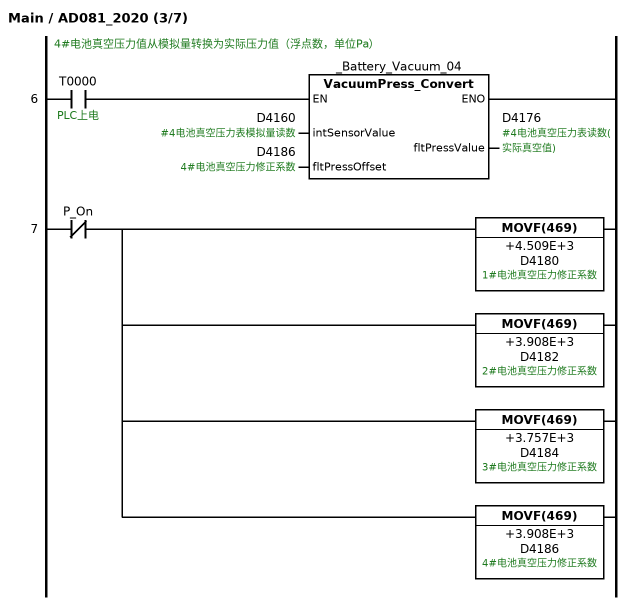
; [picture p24: Main / AD081_2020, rungs 6-7]
; rung 6: 4#电池真空压力值从模拟量转换为实际压力值（浮点数，单位Pa）
LD T0000  ; PLC上电
CALL _Battery_Vacuum_04 : VacuumPress_Convert (intSensorValue := D4160, fltPressOffset := D4186, fltPressValue => D4176)  ; #4电池真空压力表模拟量读数, 4#电池真空压力修正系数, #4电池真空压力表读数(实际真空值)
; rung 7
LDNOT P_On
MOVF(469) +4.509E+3 D4180  ; 1#电池真空压力修正系数
MOVF(469) +3.908E+3 D4182  ; 2#电池真空压力修正系数
MOVF(469) +3.757E+3 D4184  ; 3#电池真空压力修正系数
MOVF(469) +3.908E+3 D4186  ; 4#电池真空压力修正系数

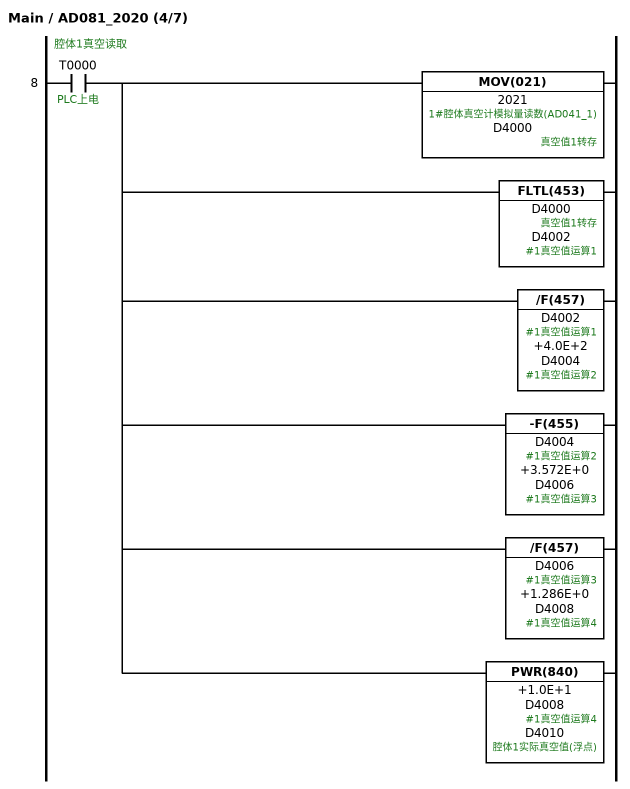
; rung 8: 腔体1真空读取
LD T0000  ; PLC上电
MOV(021) 2021 D4000  ; 1#腔体真空计模拟量读数(AD041_1), 真空值1转存
FLTL(453) D4000 D4002  ; 真空值1转存, #1真空值运算1
/F(457) D4002 +4.0E+2 D4004  ; #1真空值运算1, #1真空值运算2
-F(455) D4004 +3.572E+0 D4006  ; #1真空值运算2, #1真空值运算3
/F(457) D4006 +1.286E+0 D4008  ; #1真空值运算3, #1真空值运算4
PWR(840) +1.0E+1 D4008 D4010  ; #1真空值运算4, 腔体1实际真空值(浮点)

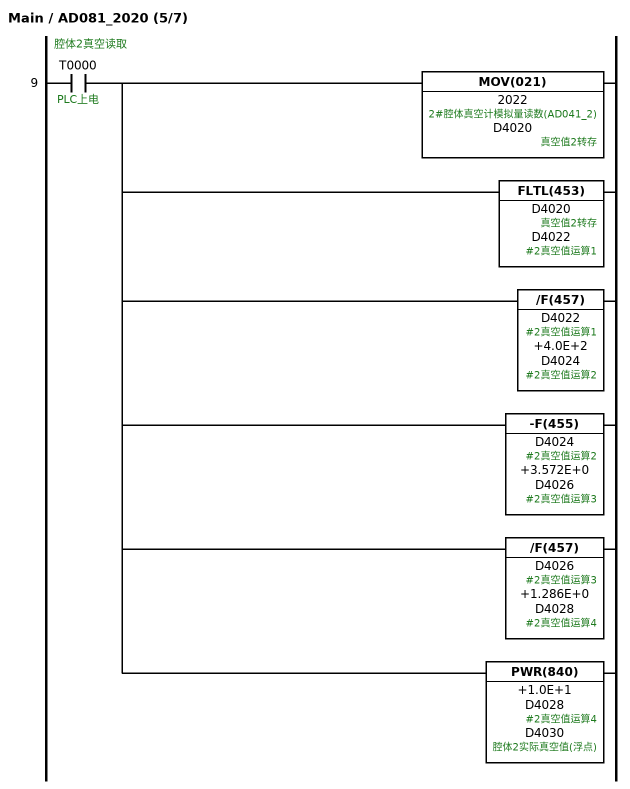
; rung 9: 腔体2真空读取
LD T0000  ; PLC上电
MOV(021) 2022 D4020  ; 2#腔体真空计模拟量读数(AD041_2), 真空值2转存
FLTL(453) D4020 D4022  ; 真空值2转存, #2真空值运算1
/F(457) D4022 +4.0E+2 D4024  ; #2真空值运算1, #2真空值运算2
-F(455) D4024 +3.572E+0 D4026  ; #2真空值运算2, #2真空值运算3
/F(457) D4026 +1.286E+0 D4028  ; #2真空值运算3, #2真空值运算4
PWR(840) +1.0E+1 D4028 D4030  ; #2真空值运算4, 腔体2实际真空值(浮点)

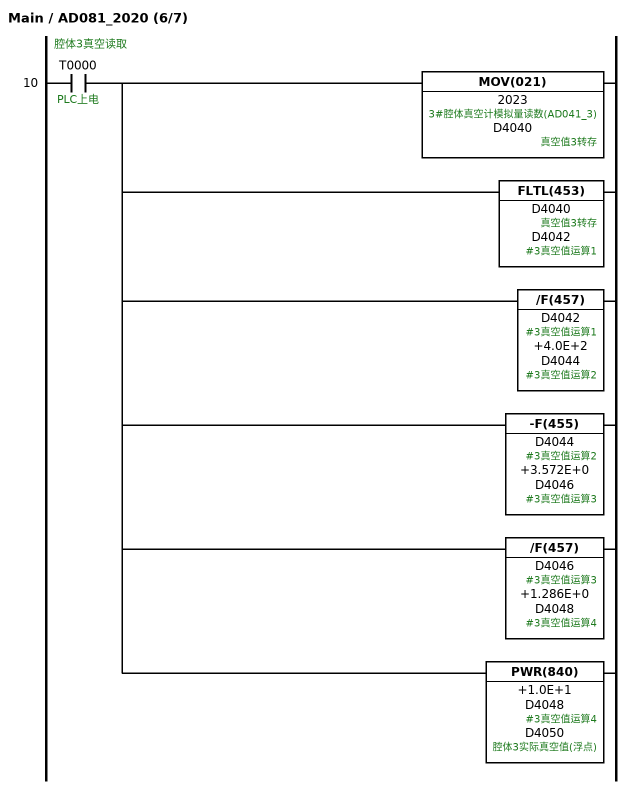
; rung 10: 腔体3真空读取
LD T0000  ; PLC上电
MOV(021) 2023 D4040  ; 3#腔体真空计模拟量读数(AD041_3), 真空值3转存
FLTL(453) D4040 D4042  ; 真空值3转存, #3真空值运算1
/F(457) D4042 +4.0E+2 D4044  ; #3真空值运算1, #3真空值运算2
-F(455) D4044 +3.572E+0 D4046  ; #3真空值运算2, #3真空值运算3
/F(457) D4046 +1.286E+0 D4048  ; #3真空值运算3, #3真空值运算4
PWR(840) +1.0E+1 D4048 D4050  ; #3真空值运算4, 腔体3实际真空值(浮点)

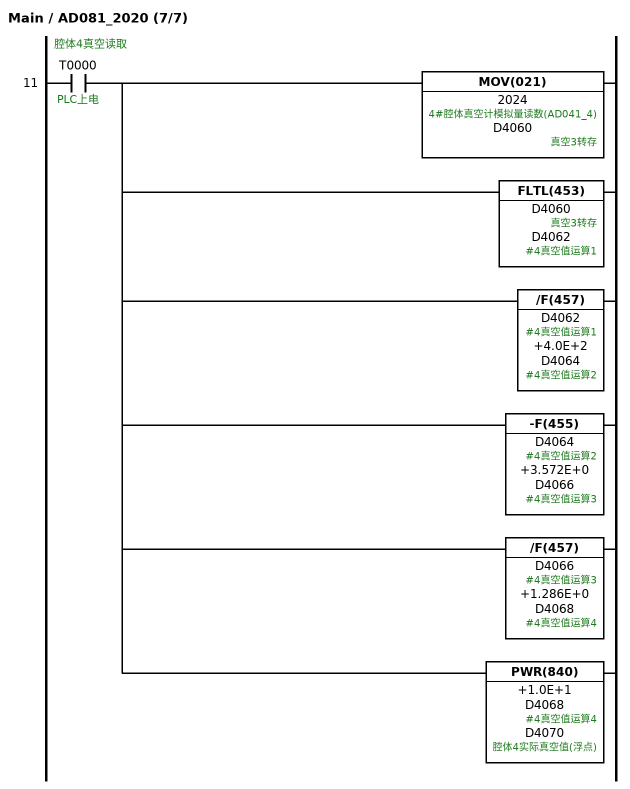
; rung 11: 腔体4真空读取
LD T0000  ; PLC上电
MOV(021) 2024 D4060  ; 4#腔体真空计模拟量读数(AD041_4), 真空3转存
FLTL(453) D4060 D4062  ; 真空3转存, #4真空值运算1
/F(457) D4062 +4.0E+2 D4064  ; #4真空值运算1, #4真空值运算2
-F(455) D4064 +3.572E+0 D4066  ; #4真空值运算2, #4真空值运算3
/F(457) D4066 +1.286E+0 D4068  ; #4真空值运算3, #4真空值运算4
PWR(840) +1.0E+1 D4068 D4070  ; #4真空值运算4, 腔体4实际真空值(浮点)

### Section 复位

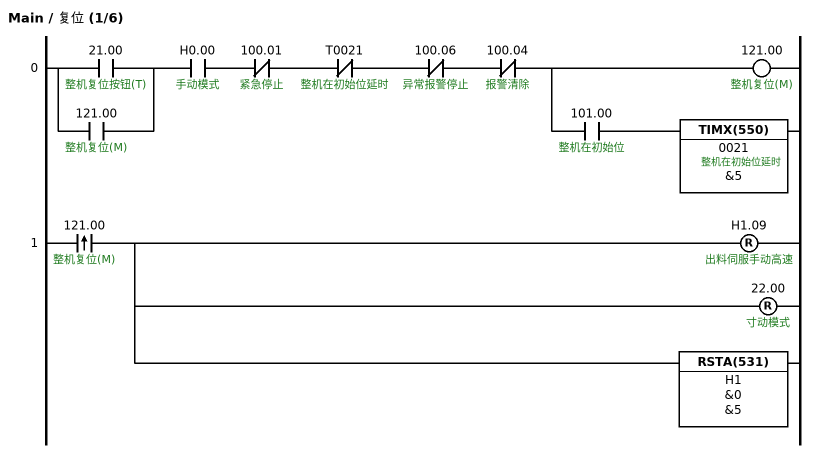
; rung 0
LD 21.00  ; 整机复位按钮(T)
OR 121.00  ; 整机复位(M)
AND H0.00  ; 手动模式
ANDNOT 100.01  ; 紧急停止
ANDNOT T0021  ; 整机在初始位延时
ANDNOT 100.06  ; 异常报警停止
ANDNOT 100.04  ; 报警清除
OUT 121.00  ; 整机复位(M)
AND 101.00  ; 整机在初始位
TIMX(550) 0021 &5  ; 整机在初始位延时
; rung 1
@LD 121.00  ; 整机复位(M)
RSET H1.09  ; 出料伺服手动高速
RSET 22.00  ; 寸动模式
RSTA(531) H1 &0 &5

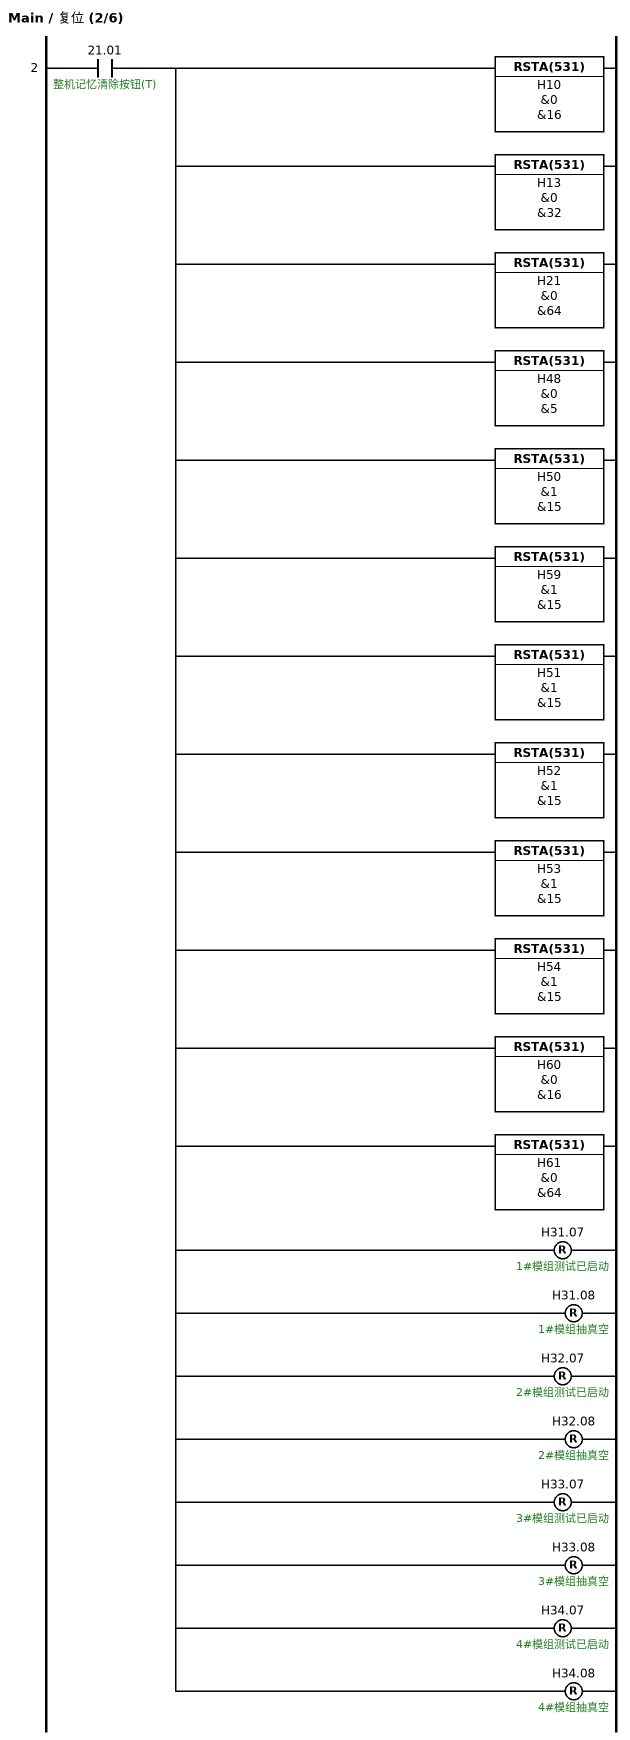
; rung 2
LD 21.01  ; 整机记忆清除按钮(T)
RSTA(531) H10 &0 &16
RSTA(531) H13 &0 &32
RSTA(531) H21 &0 &64
RSTA(531) H48 &0 &5
RSTA(531) H50 &1 &15
RSTA(531) H59 &1 &15
RSTA(531) H51 &1 &15
RSTA(531) H52 &1 &15
RSTA(531) H53 &1 &15
RSTA(531) H54 &1 &15
RSTA(531) H60 &0 &16
RSTA(531) H61 &0 &64
RSET H31.07  ; 1#模组测试已启动
RSET H31.08  ; 1#模组抽真空
RSET H32.07  ; 2#模组测试已启动
RSET H32.08  ; 2#模组抽真空
RSET H33.07  ; 3#模组测试已启动
RSET H33.08  ; 3#模组抽真空
RSET H34.07  ; 4#模组测试已启动
RSET H34.08  ; 4#模组抽真空

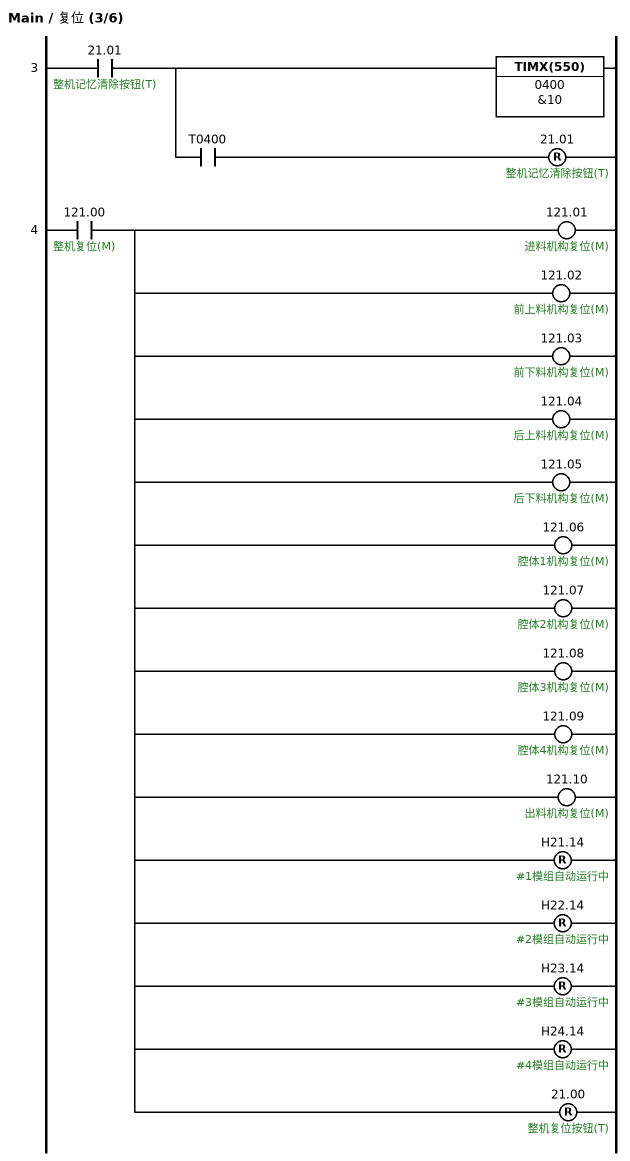
; rung 3
LD 21.01  ; 整机记忆清除按钮(T)
TIMX(550) 0400 &10
AND T0400
RSET 21.01  ; 整机记忆清除按钮(T)
; rung 4
LD 121.00  ; 整机复位(M)
OUT 121.01  ; 进料机构复位(M)
OUT 121.02  ; 前上料机构复位(M)
OUT 121.03  ; 前下料机构复位(M)
OUT 121.04  ; 后上料机构复位(M)
OUT 121.05  ; 后下料机构复位(M)
OUT 121.06  ; 腔体1机构复位(M)
OUT 121.07  ; 腔体2机构复位(M)
OUT 121.08  ; 腔体3机构复位(M)
OUT 121.09  ; 腔体4机构复位(M)
OUT 121.10  ; 出料机构复位(M)
RSET H21.14  ; #1模组自动运行中
RSET H22.14  ; #2模组自动运行中
RSET H23.14  ; #3模组自动运行中
RSET H24.14  ; #4模组自动运行中
RSET 21.00  ; 整机复位按钮(T)

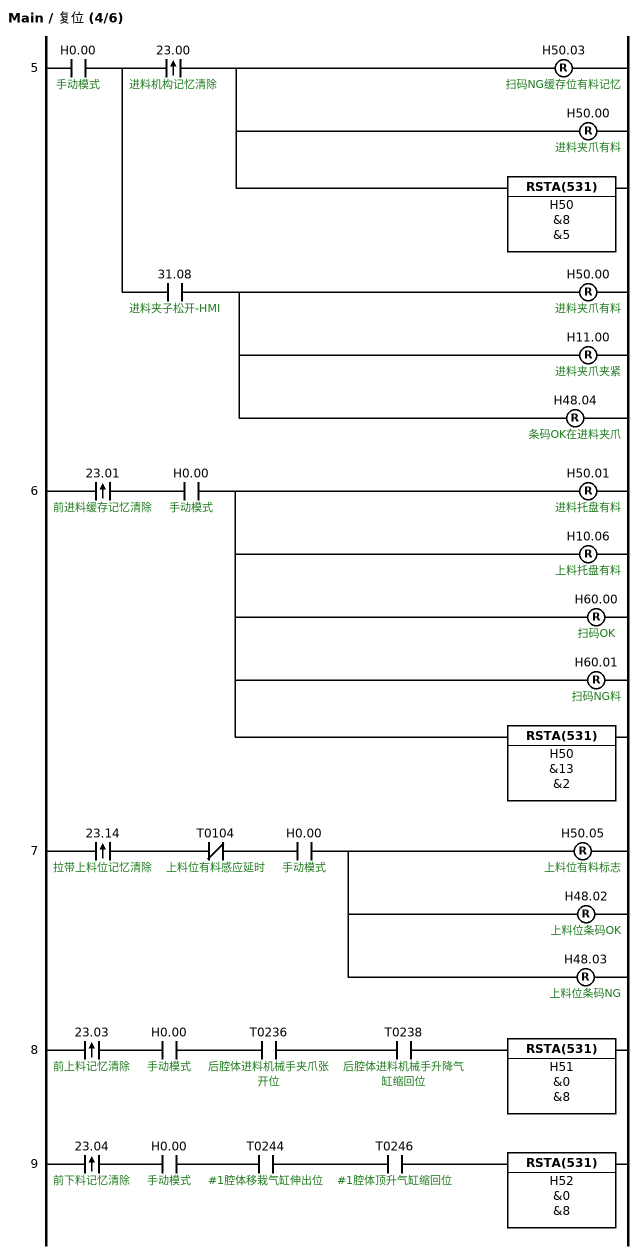
; rung 5
LD H0.00  ; 手动模式
OUT TR0
@AND 23.00  ; 进料机构记忆清除
RSET H50.03  ; 扫码NG缓存位有料记忆
RSET H50.00  ; 进料夹爪有料
RSTA(531) H50 &8 &5
LD TR0
AND 31.08  ; 进料夹子松开-HMI
RSET H50.00  ; 进料夹爪有料
RSET H11.00  ; 进料夹爪夹紧
RSET H48.04  ; 条码OK在进料夹爪
; rung 6
@LD 23.01  ; 前进料缓存记忆清除
AND H0.00  ; 手动模式
RSET H50.01  ; 进料托盘有料
RSET H10.06  ; 上料托盘有料
RSET H60.00  ; 扫码OK
RSET H60.01  ; 扫码NG料
RSTA(531) H50 &13 &2
; rung 7
@LD 23.14  ; 拉带上料位记忆清除
ANDNOT T0104  ; 上料位有料感应延时
AND H0.00  ; 手动模式
RSET H50.05  ; 上料位有料标志
RSET H48.02  ; 上料位条码OK
RSET H48.03  ; 上料位条码NG
; rung 8
@LD 23.03  ; 前上料记忆清除
AND H0.00  ; 手动模式
AND T0236  ; 后腔体进料机械手夹爪张开位
AND T0238  ; 后腔体进料机械手升降气缸缩回位
RSTA(531) H51 &0 &8
; rung 9
@LD 23.04  ; 前下料记忆清除
AND H0.00  ; 手动模式
AND T0244  ; #1腔体移栽气缸伸出位
AND T0246  ; #1腔体顶升气缸缩回位
RSTA(531) H52 &0 &8

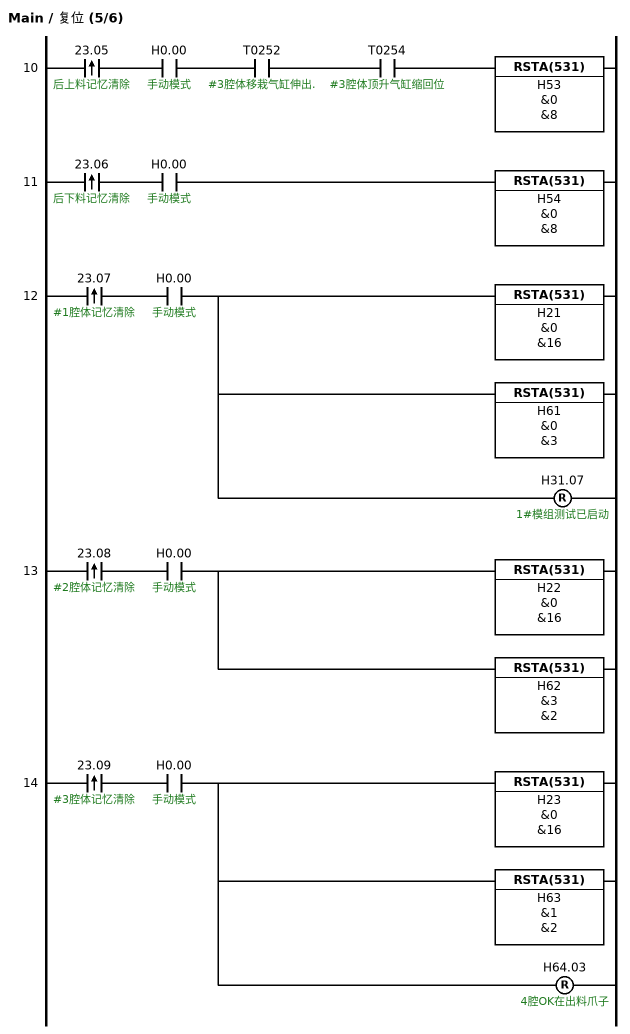
; rung 10
@LD 23.05  ; 后上料记忆清除
AND H0.00  ; 手动模式
AND T0252  ; #3腔体移栽气缸伸出.
AND T0254  ; #3腔体顶升气缸缩回位
RSTA(531) H53 &0 &8
; rung 11
@LD 23.06  ; 后下料记忆清除
AND H0.00  ; 手动模式
RSTA(531) H54 &0 &8
; rung 12
@LD 23.07  ; #1腔体记忆清除
AND H0.00  ; 手动模式
RSTA(531) H21 &0 &16
RSTA(531) H61 &0 &3
RSET H31.07  ; 1#模组测试已启动
; rung 13
@LD 23.08  ; #2腔体记忆清除
AND H0.00  ; 手动模式
RSTA(531) H22 &0 &16
RSTA(531) H62 &3 &2
; rung 14
@LD 23.09  ; #3腔体记忆清除
AND H0.00  ; 手动模式
RSTA(531) H23 &0 &16
RSTA(531) H63 &1 &2
RSET H64.03  ; 4腔OK在出料爪子

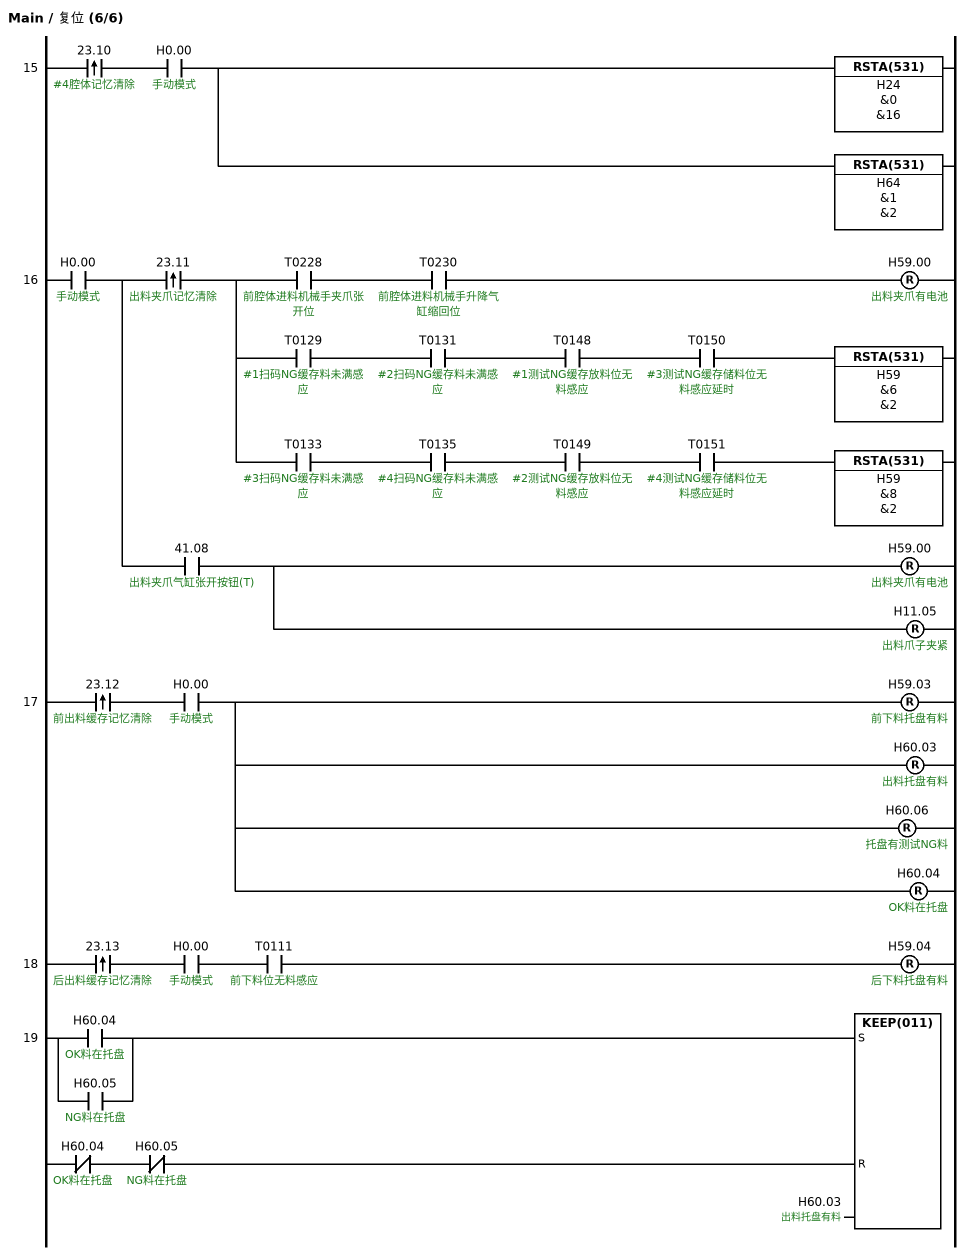
; rung 15
@LD 23.10  ; #4腔体记忆清除
AND H0.00  ; 手动模式
RSTA(531) H24 &0 &16
RSTA(531) H64 &1 &2
; rung 16
LD H0.00  ; 手动模式
OUT TR0
@AND 23.11  ; 出料夹爪记忆清除
OUT TR1
AND T0228  ; 前腔体进料机械手夹爪张开位
AND T0230  ; 前腔体进料机械手升降气缸缩回位
RSET H59.00  ; 出料夹爪有电池
LD TR1
AND T0129  ; #1扫码NG缓存料未满感应
AND T0131  ; #2扫码NG缓存料未满感应
AND T0148  ; #1测试NG缓存放料位无料感应
AND T0150  ; #3测试NG缓存储料位无料感应延时
RSTA(531) H59 &6 &2
LD TR1
AND T0133  ; #3扫码NG缓存料未满感应
AND T0135  ; #4扫码NG缓存料未满感应
AND T0149  ; #2测试NG缓存放料位无料感应
AND T0151  ; #4测试NG缓存储料位无料感应延时
RSTA(531) H59 &8 &2
LD TR0
AND 41.08  ; 出料夹爪气缸张开按钮(T)
RSET H59.00  ; 出料夹爪有电池
RSET H11.05  ; 出料爪子夹紧
; rung 17
@LD 23.12  ; 前出料缓存记忆清除
AND H0.00  ; 手动模式
RSET H59.03  ; 前下料托盘有料
RSET H60.03  ; 出料托盘有料
RSET H60.06  ; 托盘有测试NG料
RSET H60.04  ; OK料在托盘
; rung 18
@LD 23.13  ; 后出料缓存记忆清除
AND H0.00  ; 手动模式
AND T0111  ; 前下料位无料感应
RSET H59.04  ; 后下料托盘有料
; rung 19
LD H60.04  ; OK料在托盘
OR H60.05  ; NG料在托盘
LDNOT H60.04  ; OK料在托盘
ANDNOT H60.05  ; NG料在托盘
KEEP(011) H60.03  ; 出料托盘有料

### Section 外部输出

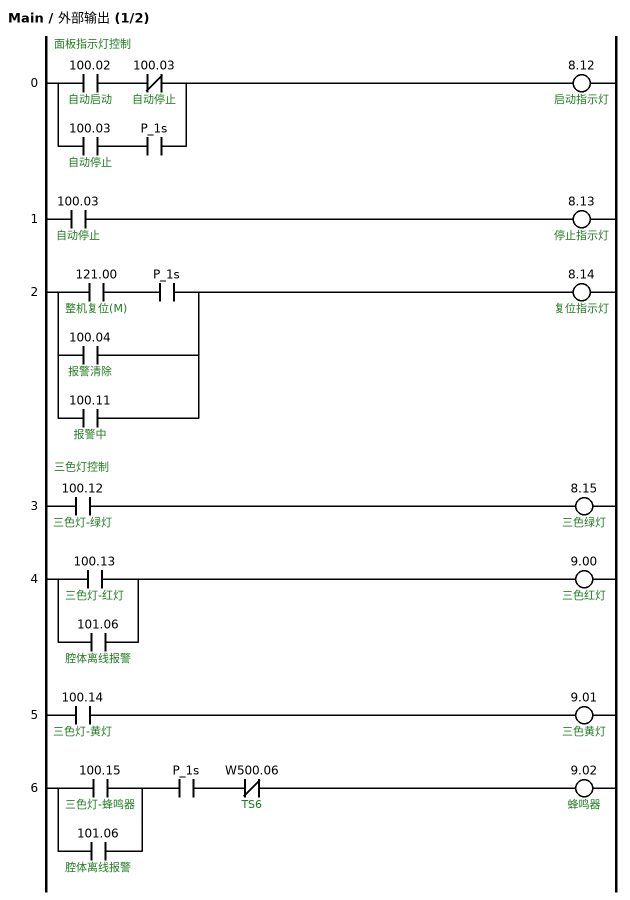
; rung 0: 面板指示灯控制
LD 100.02  ; 自动启动
ANDNOT 100.03  ; 自动停止
LD 100.03  ; 自动停止
AND P_1s
ORLD
OUT 8.12  ; 启动指示灯
; rung 1
LD 100.03  ; 自动停止
OUT 8.13  ; 停止指示灯
; rung 2
LD 121.00  ; 整机复位(M)
AND P_1s
OR 100.04  ; 报警清除
OR 100.11  ; 报警中
OUT 8.14  ; 复位指示灯
; rung 3: 三色灯控制
LD 100.12  ; 三色灯-绿灯
OUT 8.15  ; 三色绿灯
; rung 4
LD 100.13  ; 三色灯-红灯
OR 101.06  ; 腔体离线报警
OUT 9.00  ; 三色红灯
; rung 5
LD 100.14  ; 三色灯-黄灯
OUT 9.01  ; 三色黄灯
; rung 6
LD 100.15  ; 三色灯-蜂鸣器
OR 101.06  ; 腔体离线报警
AND P_1s
ANDNOT W500.06  ; TS6
OUT 9.02  ; 蜂鸣器

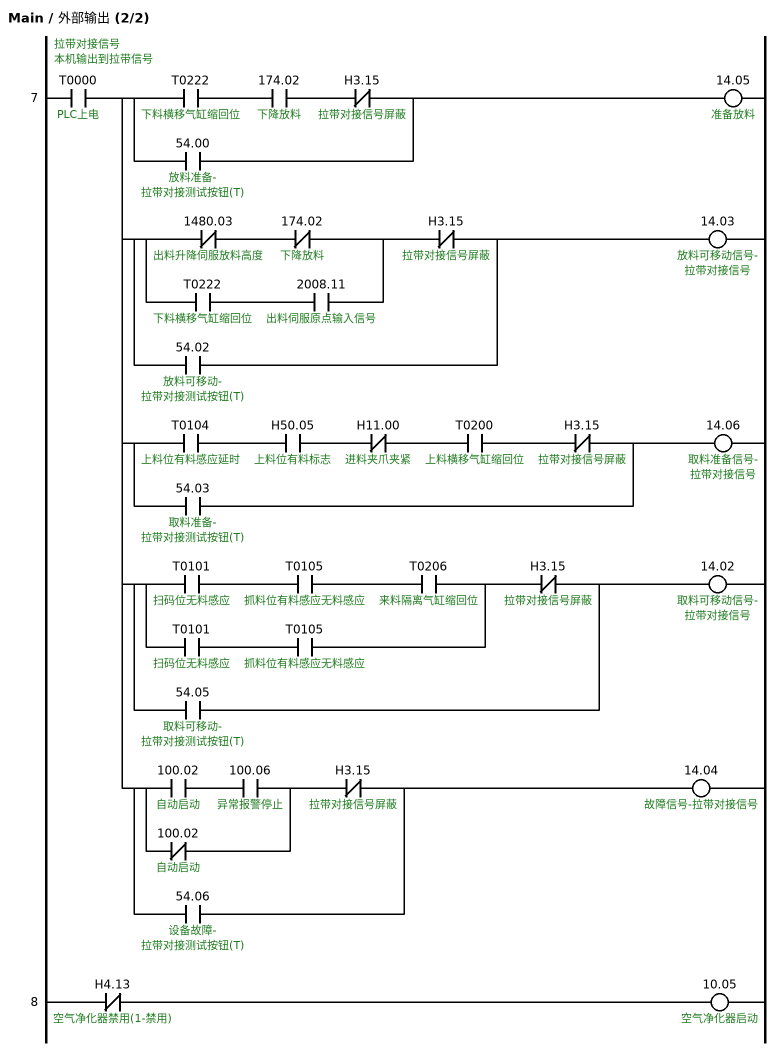
; rung 7: 拉带对接信号 / 本机输出到拉带信号
LD T0000  ; PLC上电
OUT TR0
LD T0222  ; 下料横移气缸缩回位
AND 174.02  ; 下降放料
ANDNOT H3.15  ; 拉带对接信号屏蔽
OR 54.00  ; 放料准备-拉带对接测试按钮(T)
ANDLD
OUT 14.05  ; 准备放料
LD TR0
LDNOT 1480.03  ; 出料升降伺服放料高度
ANDNOT 174.02  ; 下降放料
LD T0222  ; 下料横移气缸缩回位
AND 2008.11  ; 出料伺服原点输入信号
ORLD
ANDNOT H3.15  ; 拉带对接信号屏蔽
OR 54.02  ; 放料可移动-拉带对接测试按钮(T)
ANDLD
OUT 14.03  ; 放料可移动信号-拉带对接信号
LD TR0
LD T0104  ; 上料位有料感应延时
AND H50.05  ; 上料位有料标志
ANDNOT H11.00  ; 进料夹爪夹紧
AND T0200  ; 上料横移气缸缩回位
ANDNOT H3.15  ; 拉带对接信号屏蔽
OR 54.03  ; 取料准备-拉带对接测试按钮(T)
ANDLD
OUT 14.06  ; 取料准备信号-拉带对接信号
LD TR0
LD T0101  ; 扫码位无料感应
AND T0105  ; 抓料位有料感应无料感应
AND T0206  ; 来料隔离气缸缩回位
LD T0101  ; 扫码位无料感应
AND T0105  ; 抓料位有料感应无料感应
ORLD
ANDNOT H3.15  ; 拉带对接信号屏蔽
OR 54.05  ; 取料可移动-拉带对接测试按钮(T)
ANDLD
OUT 14.02  ; 取料可移动信号-拉带对接信号
LD TR0
LD 100.02  ; 自动启动
AND 100.06  ; 异常报警停止
ORNOT 100.02  ; 自动启动
ANDNOT H3.15  ; 拉带对接信号屏蔽
OR 54.06  ; 设备故障-拉带对接测试按钮(T)
ANDLD
OUT 14.04  ; 故障信号-拉带对接信号
; rung 8
LDNOT H4.13  ; 空气净化器禁用(1-禁用)
OUT 10.05  ; 空气净化器启动

### Section 指示灯

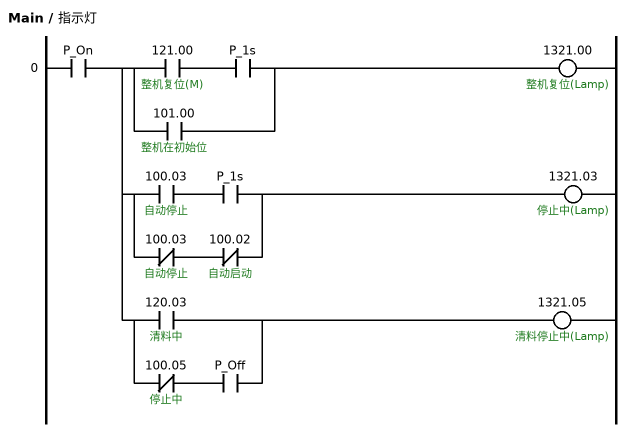
; rung 0
LD P_On
OUT TR0
LD 121.00  ; 整机复位(M)
AND P_1s
OR 101.00  ; 整机在初始位
ANDLD
OUT 1321.00  ; 整机复位(Lamp)
LD TR0
LD 100.03  ; 自动停止
AND P_1s
LDNOT 100.03  ; 自动停止
ANDNOT 100.02  ; 自动启动
ORLD
ANDLD
OUT 1321.03  ; 停止中(Lamp)
LD TR0
LD 120.03  ; 清料中
LDNOT 100.05  ; 停止中
AND P_Off
ORLD
ANDLD
OUT 1321.05  ; 清料停止中(Lamp)

### Section END
; rung 0
END(001)

## Program 进出料机构 (cyclic task 1)
Local symbols
f114 BOOL
mep BOOL

### Section Main进料

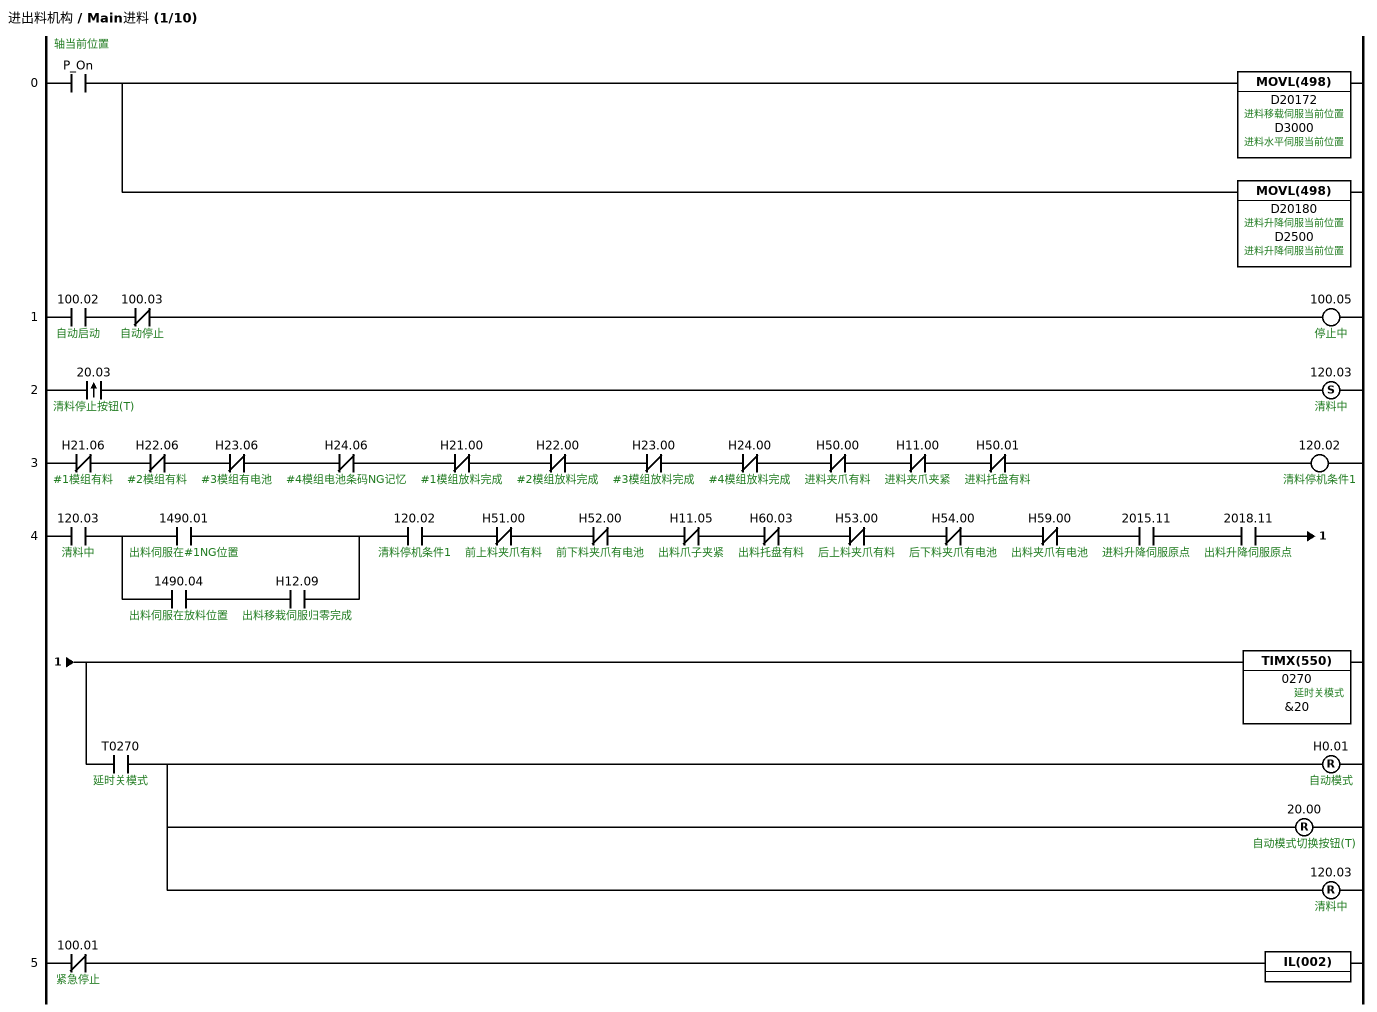
; rung 0: 轴当前位置
LD P_On
MOVL(498) D20172 D3000  ; 进料移载伺服当前位置, 进料水平伺服当前位置
MOVL(498) D20180 D2500  ; 进料升降伺服当前位置
; rung 1
LD 100.02  ; 自动启动
ANDNOT 100.03  ; 自动停止
OUT 100.05  ; 停止中
; rung 2
@LD 20.03  ; 清料停止按钮(T)
SET 120.03  ; 清料中
; rung 3
LDNOT H21.06  ; #1模组有料
ANDNOT H22.06  ; #2模组有料
ANDNOT H23.06  ; #3模组有电池
ANDNOT H24.06  ; #4模组电池条码NG记忆
ANDNOT H21.00  ; #1模组放料完成
ANDNOT H22.00  ; #2模组放料完成
ANDNOT H23.00  ; #3模组放料完成
ANDNOT H24.00  ; #4模组放料完成
ANDNOT H50.00  ; 进料夹爪有料
ANDNOT H11.00  ; 进料夹爪夹紧
ANDNOT H50.01  ; 进料托盘有料
OUT 120.02  ; 清料停机条件1
; rung 4
LD 120.03  ; 清料中
LD 1490.01  ; 出料伺服在#1NG位置
LD 1490.04  ; 出料伺服在放料位置
AND H12.09  ; 出料移栽伺服归零完成
ORLD
ANDLD
AND 120.02  ; 清料停机条件1
ANDNOT H51.00  ; 前上料夹爪有料
ANDNOT H52.00  ; 前下料夹爪有电池
ANDNOT H11.05  ; 出料爪子夹紧
ANDNOT H60.03  ; 出料托盘有料
ANDNOT H53.00  ; 后上料夹爪有料
ANDNOT H54.00  ; 后下料夹爪有电池
ANDNOT H59.00  ; 出料夹爪有电池
AND 2015.11  ; 进料升降伺服原点
AND 2018.11  ; 出料升降伺服原点
TIMX(550) 0270 &20  ; 延时关模式
AND T0270  ; 延时关模式
RSET H0.01  ; 自动模式
RSET 20.00  ; 自动模式切换按钮(T)
RSET 120.03  ; 清料中
; rung 5
LDNOT 100.01  ; 紧急停止
IL(002)

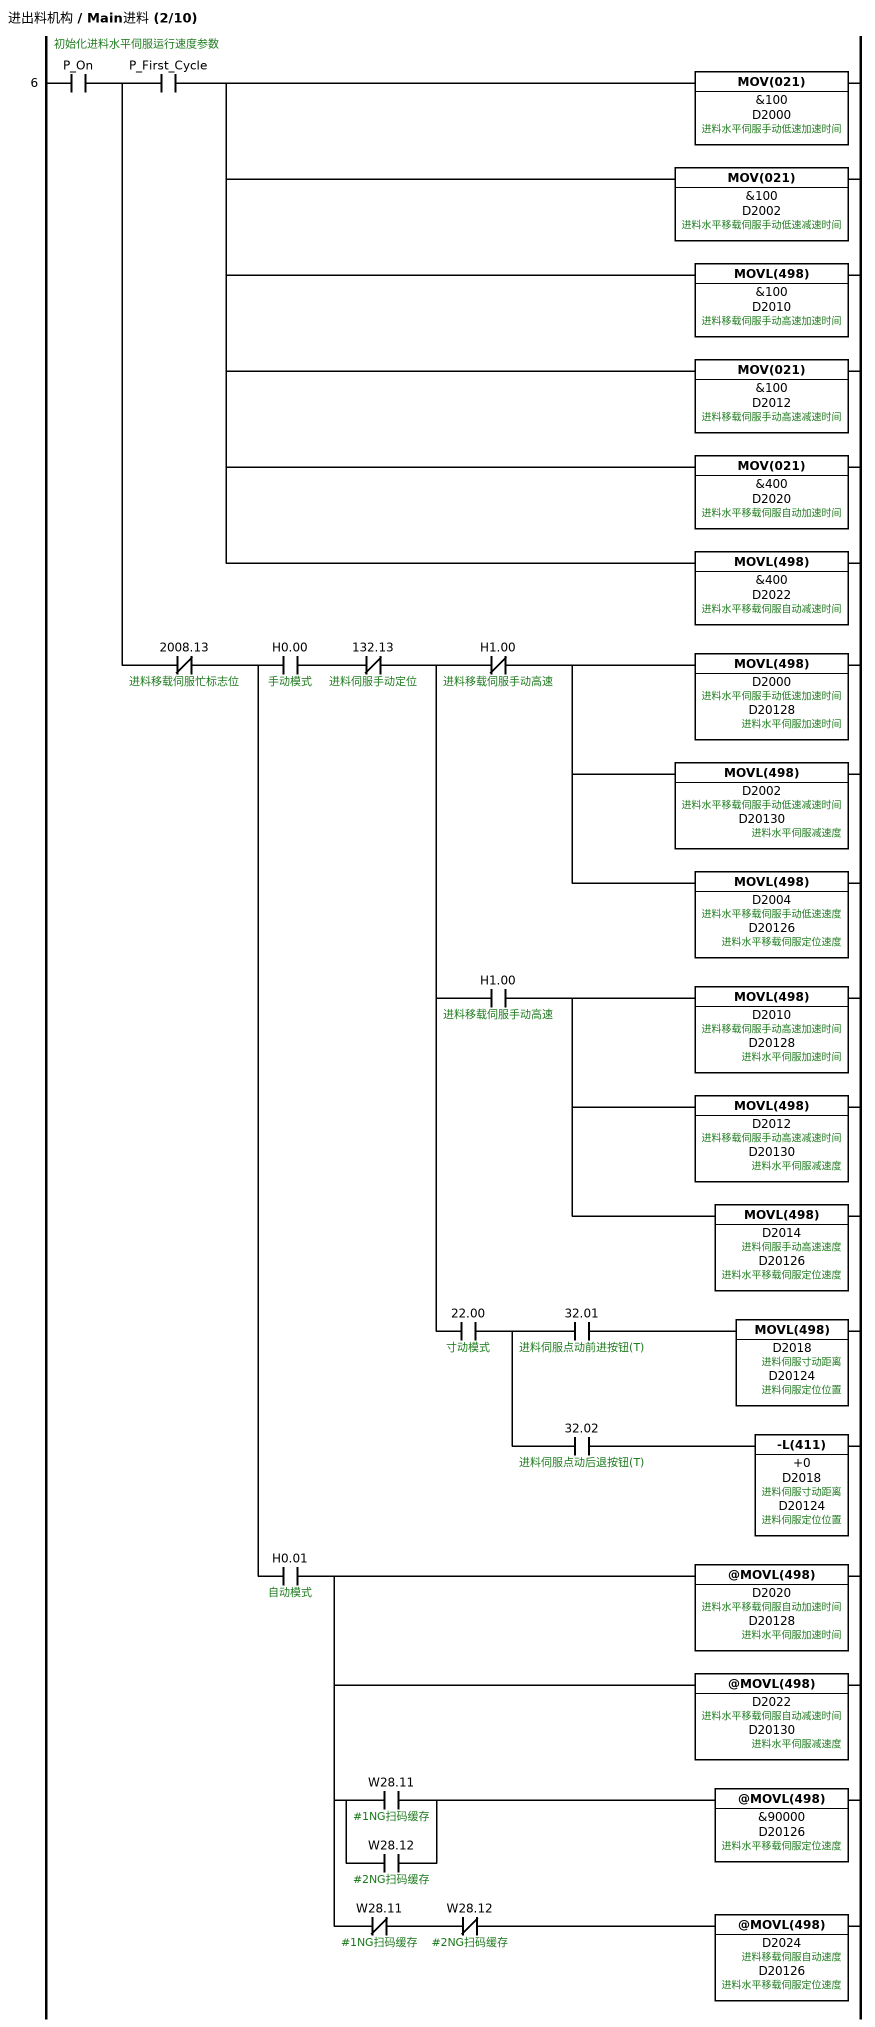
; rung 6: 初始化进料水平伺服运行速度参数
LD P_On
OUT TR0
AND P_First_Cycle
MOV(021) &100 D2000  ; 进料水平伺服手动低速加速时间
MOV(021) &100 D2002  ; 进料水平移载伺服手动低速减速时间
MOVL(498) &100 D2010  ; 进料移载伺服手动高速加速时间
MOV(021) &100 D2012  ; 进料移载伺服手动高速减速时间
MOV(021) &400 D2020  ; 进料水平移载伺服自动加速时间
MOVL(498) &400 D2022  ; 进料水平移载伺服自动减速时间
LD TR0
ANDNOT 2008.13  ; 进料移载伺服忙标志位
OUT TR0
AND H0.00  ; 手动模式
ANDNOT 132.13  ; 进料伺服手动定位
OUT TR1
ANDNOT H1.00  ; 进料移载伺服手动高速
MOVL(498) D2000 D20128  ; 进料水平伺服手动低速加速时间, 进料水平伺服加速时间
MOVL(498) D2002 D20130  ; 进料水平移载伺服手动低速减速时间, 进料水平伺服减速度
MOVL(498) D2004 D20126  ; 进料水平移载伺服手动低速速度, 进料水平移载伺服定位速度
LD TR1
AND H1.00  ; 进料移载伺服手动高速
MOVL(498) D2010 D20128  ; 进料移载伺服手动高速加速时间, 进料水平伺服加速时间
MOVL(498) D2012 D20130  ; 进料移载伺服手动高速减速时间, 进料水平伺服减速度
MOVL(498) D2014 D20126  ; 进料伺服手动高速速度, 进料水平移载伺服定位速度
LD TR1
AND 22.00  ; 寸动模式
OUT TR1
AND 32.01  ; 进料伺服点动前进按钮(T)
MOVL(498) D2018 D20124  ; 进料伺服寸动距离, 进料伺服定位位置
LD TR1
AND 32.02  ; 进料伺服点动后退按钮(T)
-L(411) +0 D2018 D20124  ; 进料伺服寸动距离, 进料伺服定位位置
LD TR0
AND H0.01  ; 自动模式
OUT TR0
@MOVL(498) D2020 D20128  ; 进料水平移载伺服自动加速时间, 进料水平伺服加速时间
@MOVL(498) D2022 D20130  ; 进料水平移载伺服自动减速时间, 进料水平伺服减速度
LD W28.11  ; #1NG扫码缓存
OR W28.12  ; #2NG扫码缓存
ANDLD
@MOVL(498) &90000 D20126  ; 进料水平移载伺服定位速度
LD TR0
ANDNOT W28.11  ; #1NG扫码缓存
ANDNOT W28.12  ; #2NG扫码缓存
@MOVL(498) D2024 D20126  ; 进料移载伺服自动速度, 进料水平移载伺服定位速度

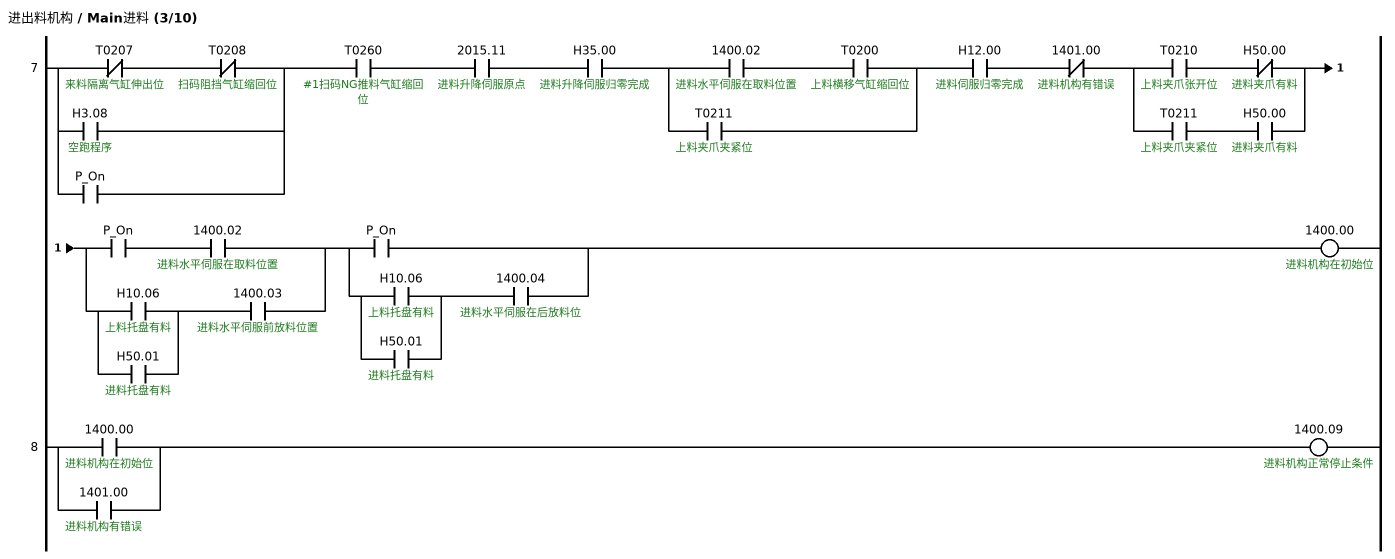
; rung 7
LDNOT T0207  ; 来料隔离气缸伸出位
ANDNOT T0208  ; 扫码阻挡气缸缩回位
OR H3.08  ; 空跑程序
OR P_On
AND T0260  ; #1扫码NG推料气缸缩回位
AND 2015.11  ; 进料升降伺服原点
AND H35.00  ; 进料升降伺服归零完成
LD 1400.02  ; 进料水平伺服在取料位置
AND T0200  ; 上料横移气缸缩回位
OR T0211  ; 上料夹爪夹紧位
ANDLD
AND H12.00  ; 进料伺服归零完成
ANDNOT 1401.00  ; 进料机构有错误
LD T0210  ; 上料夹爪张开位
ANDNOT H50.00  ; 进料夹爪有料
LD T0211  ; 上料夹爪夹紧位
AND H50.00  ; 进料夹爪有料
ORLD
ANDLD
LD P_On
AND 1400.02  ; 进料水平伺服在取料位置
LD H10.06  ; 上料托盘有料
OR H50.01  ; 进料托盘有料
AND 1400.03  ; 进料水平伺服前放料位置
ORLD
ANDLD
LD P_On
LD H10.06  ; 上料托盘有料
OR H50.01  ; 进料托盘有料
AND 1400.04  ; 进料水平伺服在后放料位
ORLD
ANDLD
OUT 1400.00  ; 进料机构在初始位
; rung 8
LD 1400.00  ; 进料机构在初始位
OR 1401.00  ; 进料机构有错误
OUT 1400.09  ; 进料机构正常停止条件

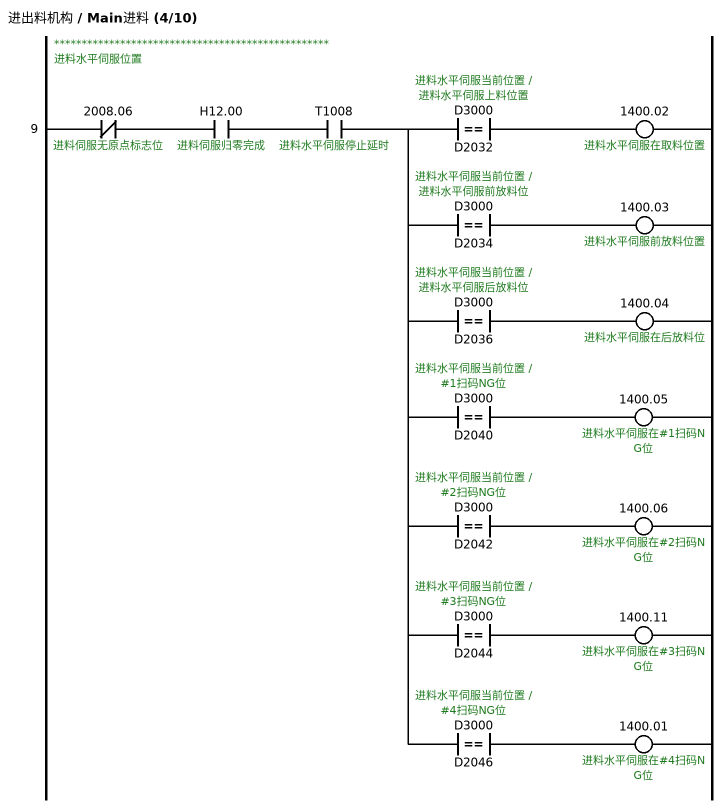
; rung 9: ************************************************** / 进料水平伺服位置
LDNOT 2008.06  ; 进料伺服无原点标志位
AND H12.00  ; 进料伺服归零完成
AND T1008  ; 进料水平伺服停止延时
OUT TR0
AND=SL(303) D3000 D2032  ; 进料水平伺服当前位置, 进料水平伺服上料位置
OUT 1400.02  ; 进料水平伺服在取料位置
LD TR0
AND=SL(303) D3000 D2034  ; 进料水平伺服当前位置, 进料水平伺服前放料位
OUT 1400.03  ; 进料水平伺服前放料位置
LD TR0
AND=SL(303) D3000 D2036  ; 进料水平伺服当前位置, 进料水平伺服后放料位
OUT 1400.04  ; 进料水平伺服在后放料位
LD TR0
AND=SL(303) D3000 D2040  ; 进料水平伺服当前位置, #1扫码NG位
OUT 1400.05  ; 进料水平伺服在#1扫码NG位
LD TR0
AND=SL(303) D3000 D2042  ; 进料水平伺服当前位置, #2扫码NG位
OUT 1400.06  ; 进料水平伺服在#2扫码NG位
LD TR0
AND=SL(303) D3000 D2044  ; 进料水平伺服当前位置, #3扫码NG位
OUT 1400.11  ; 进料水平伺服在#3扫码NG位
LD TR0
AND=SL(303) D3000 D2046  ; 进料水平伺服当前位置, #4扫码NG位
OUT 1400.01  ; 进料水平伺服在#4扫码NG位

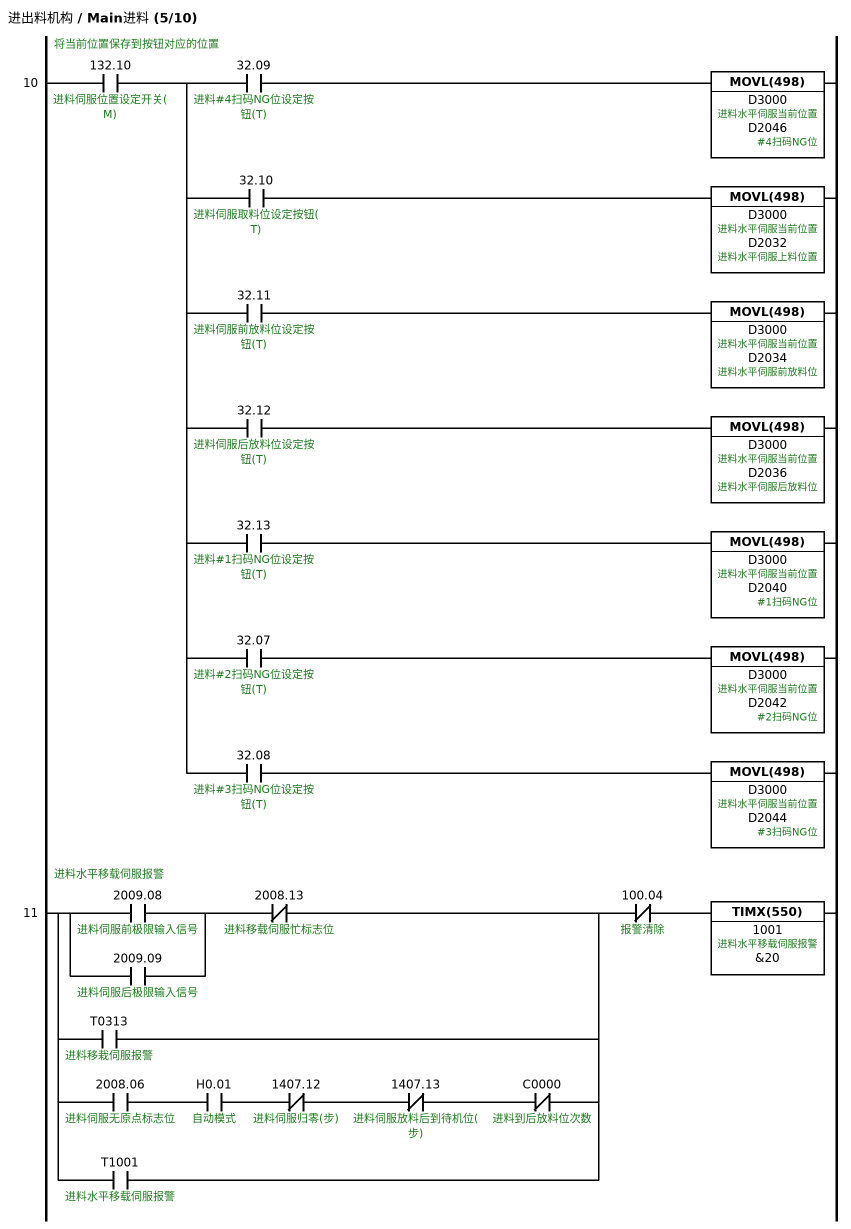
; rung 10: 将当前位置保存到按钮对应的位置
LD 132.10  ; 进料伺服位置设定开关(M)
OUT TR0
AND 32.09  ; 进料#4扫码NG位设定按钮(T)
MOVL(498) D3000 D2046  ; 进料水平伺服当前位置, #4扫码NG位
LD TR0
AND 32.10  ; 进料伺服取料位设定按钮(T)
MOVL(498) D3000 D2032  ; 进料水平伺服当前位置, 进料水平伺服上料位置
LD TR0
AND 32.11  ; 进料伺服前放料位设定按钮(T)
MOVL(498) D3000 D2034  ; 进料水平伺服当前位置, 进料水平伺服前放料位
LD TR0
AND 32.12  ; 进料伺服后放料位设定按钮(T)
MOVL(498) D3000 D2036  ; 进料水平伺服当前位置, 进料水平伺服后放料位
LD TR0
AND 32.13  ; 进料#1扫码NG位设定按钮(T)
MOVL(498) D3000 D2040  ; 进料水平伺服当前位置, #1扫码NG位
LD TR0
AND 32.07  ; 进料#2扫码NG位设定按钮(T)
MOVL(498) D3000 D2042  ; 进料水平伺服当前位置, #2扫码NG位
LD TR0
AND 32.08  ; 进料#3扫码NG位设定按钮(T)
MOVL(498) D3000 D2044  ; 进料水平伺服当前位置, #3扫码NG位
; rung 11: 进料水平移载伺服报警
LD 2009.08  ; 进料伺服前极限输入信号
OR 2009.09  ; 进料伺服后极限输入信号
ANDNOT 2008.13  ; 进料移载伺服忙标志位
OR T0313  ; 进料移栽伺服报警
LD 2008.06  ; 进料伺服无原点标志位
AND H0.01  ; 自动模式
ANDNOT 1407.12  ; 进料伺服归零(步)
ANDNOT 1407.13  ; 进料伺服放料后到待机位(步)
ANDNOT C0000  ; 进料到后放料位次数
ORLD
OR T1001  ; 进料水平移载伺服报警
ANDNOT 100.04  ; 报警清除
TIMX(550) 1001 &20  ; 进料水平移载伺服报警

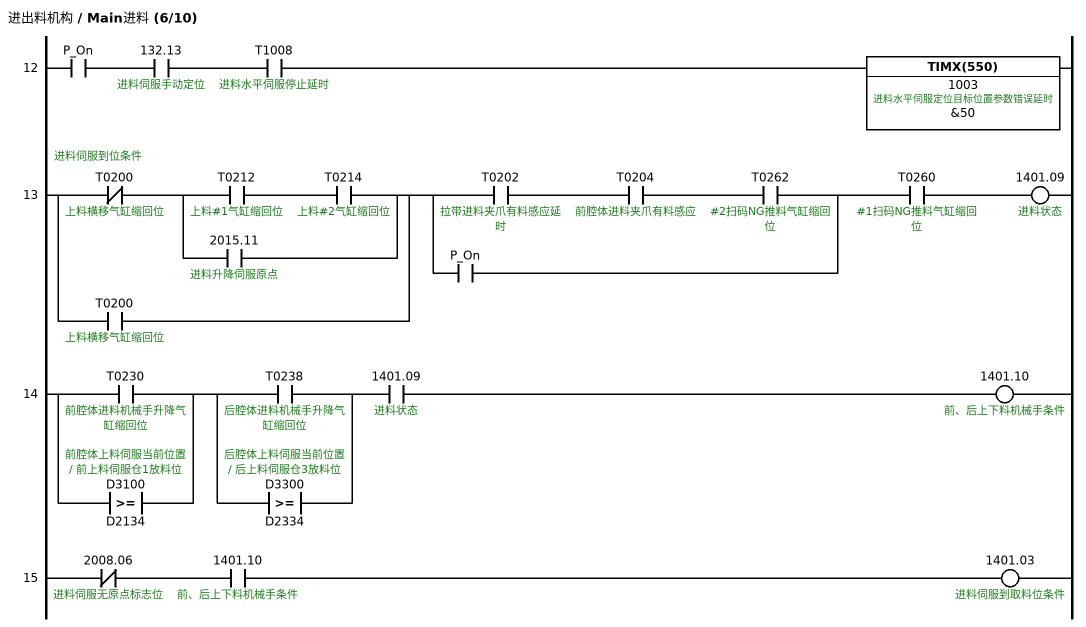
; rung 12
LD P_On
AND 132.13  ; 进料伺服手动定位
AND T1008  ; 进料水平伺服停止延时
TIMX(550) 1003 &50  ; 进料水平伺服定位目标位置参数错误延时
; rung 13: 进料伺服到位条件
LDNOT T0200  ; 上料横移气缸缩回位
LD T0212  ; 上料#1气缸缩回位
AND T0214  ; 上料#2气缸缩回位
OR 2015.11  ; 进料升降伺服原点
ANDLD
OR T0200  ; 上料横移气缸缩回位
LD T0202  ; 拉带进料夹爪有料感应延时
AND T0204  ; 前腔体进料夹爪有料感应
AND T0262  ; #2扫码NG推料气缸缩回位
OR P_On
ANDLD
AND T0260  ; #1扫码NG推料气缸缩回位
OUT 1401.09  ; 进料状态
; rung 14
LD T0230  ; 前腔体进料机械手升降气缸缩回位
OR>=SL(328) D3100 D2134  ; 前腔体上料伺服当前位置, 前上料伺服仓1放料位
LD T0238  ; 后腔体进料机械手升降气缸缩回位
OR>=SL(328) D3300 D2334  ; 后腔体上料伺服当前位置, 后上料伺服仓3放料位
ANDLD
AND 1401.09  ; 进料状态
OUT 1401.10  ; 前、后上下料机械手条件
; rung 15
LDNOT 2008.06  ; 进料伺服无原点标志位
AND 1401.10  ; 前、后上下料机械手条件
OUT 1401.03  ; 进料伺服到取料位条件

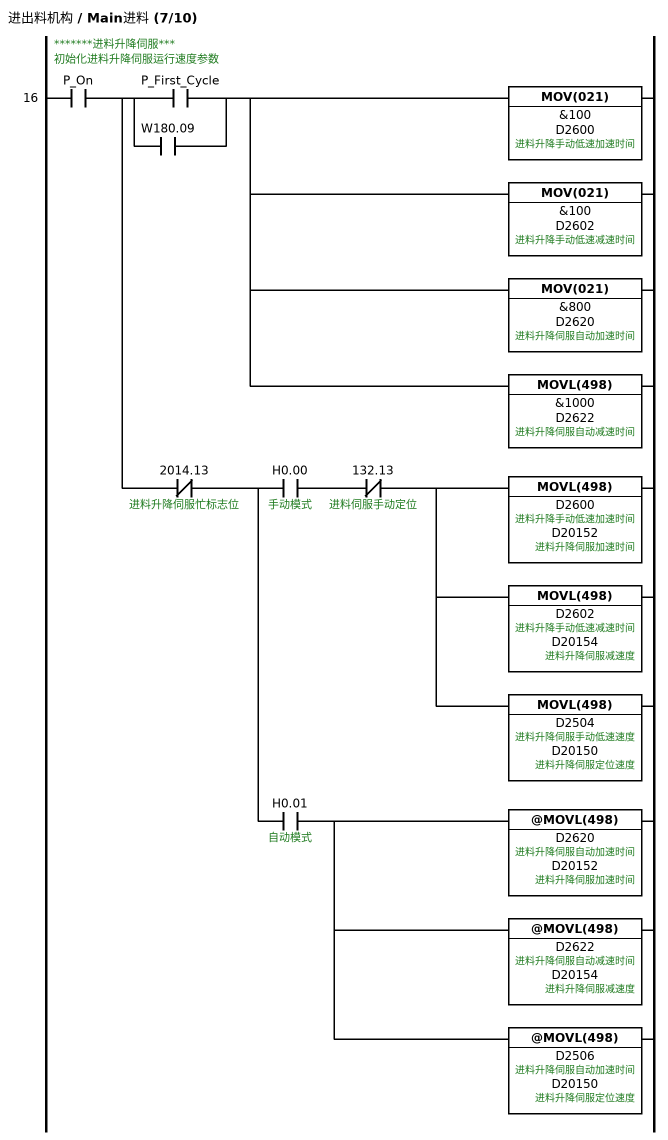
; rung 16: *******进料升降伺服*** / 初始化进料升降伺服运行速度参数
LD P_On
OUT TR0
LD P_First_Cycle
OR W180.09
ANDLD
MOV(021) &100 D2600  ; 进料升降手动低速加速时间
MOV(021) &100 D2602  ; 进料升降手动低速减速时间
MOV(021) &800 D2620  ; 进料升降伺服自动加速时间
MOVL(498) &1000 D2622  ; 进料升降伺服自动减速时间
LD TR0
ANDNOT 2014.13  ; 进料升降伺服忙标志位
OUT TR0
AND H0.00  ; 手动模式
ANDNOT 132.13  ; 进料伺服手动定位
MOVL(498) D2600 D20152  ; 进料升降手动低速加速时间, 进料升降伺服加速时间
MOVL(498) D2602 D20154  ; 进料升降手动低速减速时间, 进料升降伺服减速度
MOVL(498) D2504 D20150  ; 进料升降伺服手动低速速度, 进料升降伺服定位速度
LD TR0
AND H0.01  ; 自动模式
@MOVL(498) D2620 D20152  ; 进料升降伺服自动加速时间, 进料升降伺服加速时间
@MOVL(498) D2622 D20154  ; 进料升降伺服自动减速时间, 进料升降伺服减速度
@MOVL(498) D2506 D20150  ; 进料升降伺服自动加速时间, 进料升降伺服定位速度

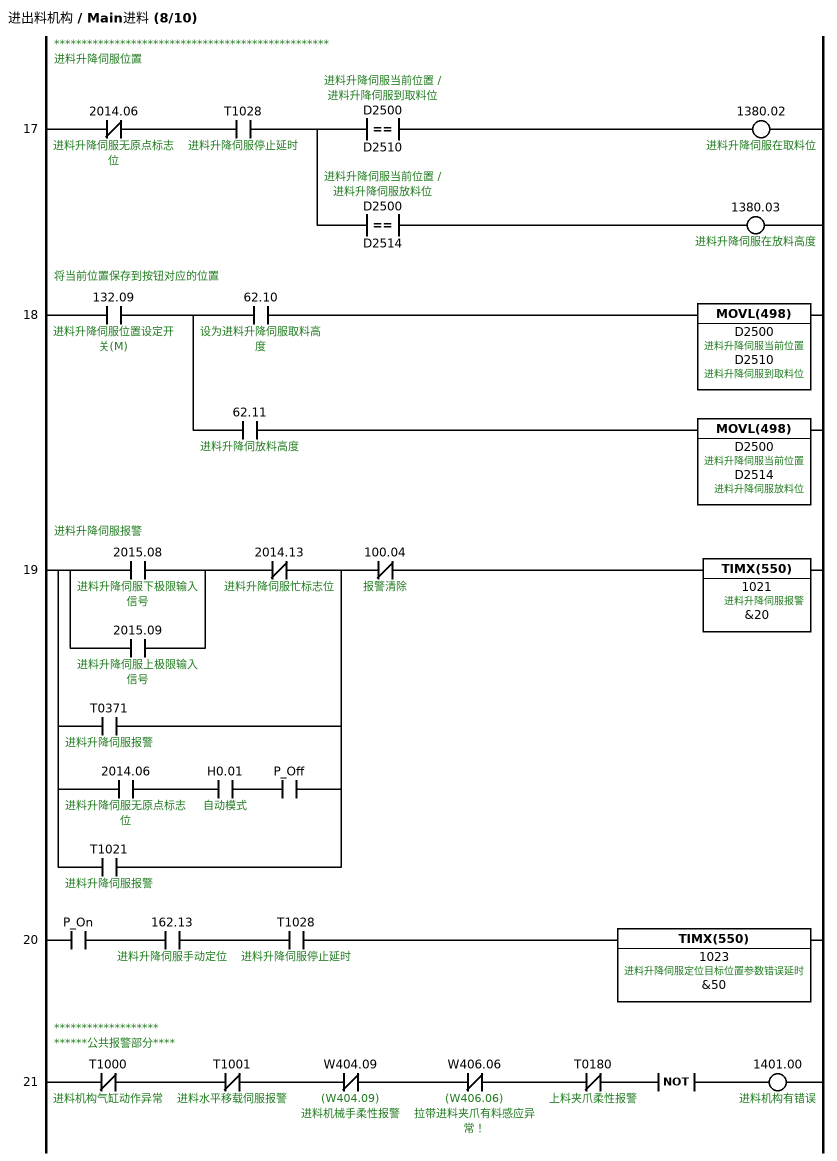
; rung 17: ************************************************** / 进料升降伺服位置
LDNOT 2014.06  ; 进料升降伺服无原点标志位
AND T1028  ; 进料升降伺服停止延时
OUT TR0
AND=SL(303) D2500 D2510  ; 进料升降伺服当前位置, 进料升降伺服到取料位
OUT 1380.02  ; 进料升降伺服在取料位
LD TR0
AND=SL(303) D2500 D2514  ; 进料升降伺服当前位置, 进料升降伺服放料位
OUT 1380.03  ; 进料升降伺服在放料高度
; rung 18: 将当前位置保存到按钮对应的位置
LD 132.09  ; 进料升降伺服位置设定开关(M)
OUT TR0
AND 62.10  ; 设为进料升降伺服取料高度
MOVL(498) D2500 D2510  ; 进料升降伺服当前位置, 进料升降伺服到取料位
LD TR0
AND 62.11  ; 进料升降伺放料高度
MOVL(498) D2500 D2514  ; 进料升降伺服当前位置, 进料升降伺服放料位
; rung 19: 进料升降伺服报警
LD 2015.08  ; 进料升降伺服下极限输入信号
OR 2015.09  ; 进料升降伺服上极限输入信号
ANDNOT 2014.13  ; 进料升降伺服忙标志位
OR T0371  ; 进料升降伺服报警
LD 2014.06  ; 进料升降伺服无原点标志位
AND H0.01  ; 自动模式
AND P_Off
ORLD
OR T1021  ; 进料升降伺服报警
ANDNOT 100.04  ; 报警清除
TIMX(550) 1021 &20  ; 进料升降伺服报警
; rung 20
LD P_On
AND 162.13  ; 进料升降伺服手动定位
AND T1028  ; 进料升降伺服停止延时
TIMX(550) 1023 &50  ; 进料升降伺服定位目标位置参数错误延时
; rung 21: ******************* / ******公共报警部分****
LDNOT T1000  ; 进料机构气缸动作异常
ANDNOT T1001  ; 进料水平移载伺服报警
ANDNOT W404.09  ; (W404.09) 进料机械手柔性报警
ANDNOT W406.06  ; (W406.06) 拉带进料夹爪有料感应异常！
ANDNOT T0180  ; 上料夹爪柔性报警
NOT(520)
OUT 1401.00  ; 进料机构有错误

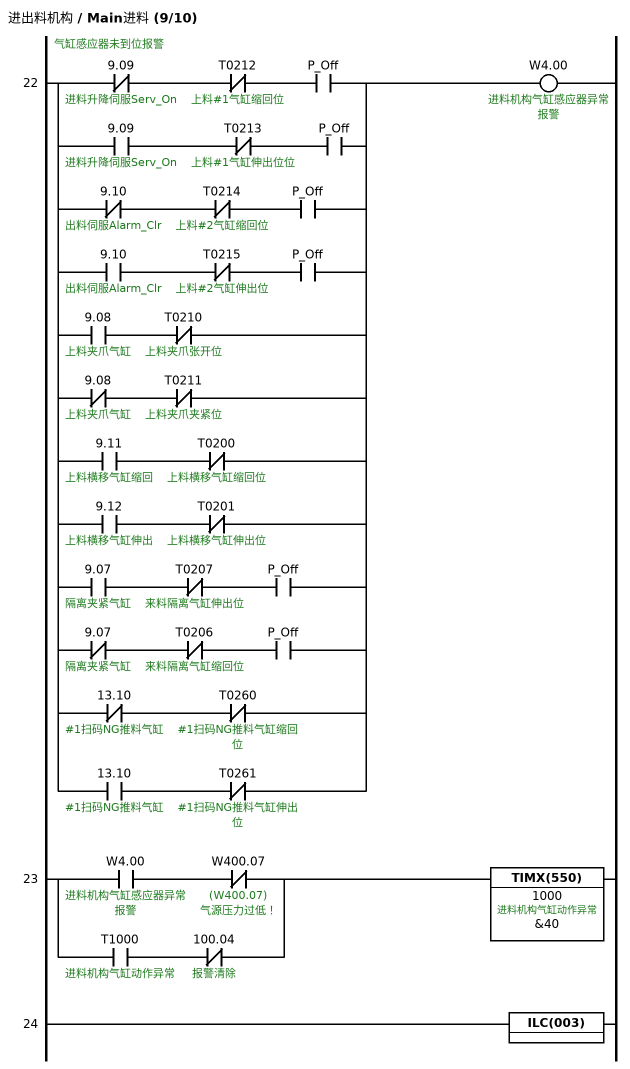
; rung 22: 气缸感应器未到位报警
LDNOT 9.09  ; 进料升降伺服Serv_On
ANDNOT T0212  ; 上料#1气缸缩回位
AND P_Off
LD 9.09  ; 进料升降伺服Serv_On
ANDNOT T0213  ; 上料#1气缸伸出位位
AND P_Off
ORLD
LDNOT 9.10  ; 出料伺服Alarm_Clr
ANDNOT T0214  ; 上料#2气缸缩回位
AND P_Off
ORLD
LD 9.10  ; 出料伺服Alarm_Clr
ANDNOT T0215  ; 上料#2气缸伸出位
AND P_Off
ORLD
LD 9.08  ; 上料夹爪气缸
ANDNOT T0210  ; 上料夹爪张开位
ORLD
LDNOT 9.08  ; 上料夹爪气缸
ANDNOT T0211  ; 上料夹爪夹紧位
ORLD
LD 9.11  ; 上料横移气缸缩回
ANDNOT T0200  ; 上料横移气缸缩回位
ORLD
LD 9.12  ; 上料横移气缸伸出
ANDNOT T0201  ; 上料横移气缸伸出位
ORLD
LD 9.07  ; 隔离夹紧气缸
ANDNOT T0207  ; 来料隔离气缸伸出位
AND P_Off
ORLD
LDNOT 9.07  ; 隔离夹紧气缸
ANDNOT T0206  ; 来料隔离气缸缩回位
AND P_Off
ORLD
LDNOT 13.10  ; #1扫码NG推料气缸
ANDNOT T0260  ; #1扫码NG推料气缸缩回位
ORLD
LD 13.10  ; #1扫码NG推料气缸
ANDNOT T0261  ; #1扫码NG推料气缸伸出位
ORLD
OUT W4.00  ; 进料机构气缸感应器异常报警
; rung 23
LD W4.00  ; 进料机构气缸感应器异常报警
ANDNOT W400.07  ; (W400.07) 气源压力过低！
LD T1000  ; 进料机构气缸动作异常
ANDNOT 100.04  ; 报警清除
ORLD
TIMX(550) 1000 &40  ; 进料机构气缸动作异常
; rung 24
ILC(003)

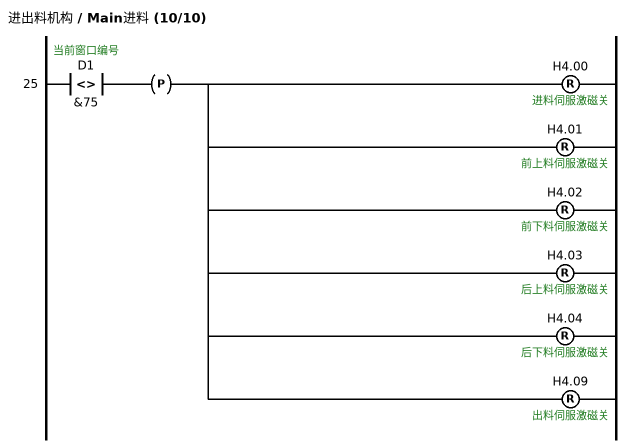
; rung 25
LD<>(305) D1 &75  ; 当前窗口编号
UP(521)
RSET H4.00  ; 进料伺服激磁关
RSET H4.01  ; 前上料伺服激磁关
RSET H4.02  ; 前下料伺服激磁关
RSET H4.03  ; 后上料伺服激磁关
RSET H4.04  ; 后下料伺服激磁关
RSET H4.09  ; 出料伺服激磁关

### Section Main出料

